# B&R Automation Studio project BR_Lab4
Automation Studio 4.5.2.102

## Configuration Real

### Task classes (Cpu.sw)
```
Cyclic#1:
  SDCAxisCtr <- SDCAxisCtrl_X.prg
DataObjects: Arnc0sys
NcDataObjects: gAxis01a <- gAxis01obj.gAxis01a.dob, gAxis01i <- gAxis01obj.gAxis01i.dob
Binaries: TCData, Acp10map1, acp10cfg, Acp10map, arconfig, User, Role, sysconf, iomap, asfw, ashwd, arnc0cfg, Arnc0map
Libraries: Acp10sdc, Library, Acp10man, Acp10_MC, sys_lib, brsystem, asstring, powerlnk, asieccon, AsMath, Arnc0man, DataObj, AsArLog, FileIO, AsArProf, AsMem, Runtime, astime, Acp10par, NcGlobal, asiotime
```

### IoMap.iom - 4PP065_0571_P74/IoMap.iom
```iecst
VAR_CONFIG
	::SDCAxisCtr:pwm_period AT %QW."X20MM4456".PeriodDurationPWM;
	::SDCAxisCtr:coil_pwm_value AT %QW."X20MM4456".PulseWidthCurrentPWM04;
	::SDCAxisCtr:axis_X.pwm_value AT %QW."X20MM4456".PulseWidthCurrentPWM01;
	::SDCAxisCtr:axis_X.reset_error AT %QX."X20MM4456".ClearError01;
	::SDCAxisCtr:axis_X.reset_counter AT %QX."X20MM4456".ResetCounter01;
	::SDCAxisCtr:axis_X.counter AT %IW."X20MM4456".Counter01;
	::SDCAxisCtr:coil_powered AT %IX."X20DI9371".DigitalInput01;
	::SDCAxisCtr:axis_X.endswitch_a_reached AT %IX."X20MM4456".StatusInput03;
	::SDCAxisCtr:axis_X.endswitch_b_reached AT %IX."X20MM4456".StatusInput04;
	::SDCAxisCtr:posEnable.enable AT %IX."X20DI9371".DigitalInput02; (*Insert your comment here...*)
	::SDCAxisCtr:posEnableRight.enable AT %IX."X20DI9371".DigitalInput03; (*Insert your comment here...*)
END_VAR
```

## Logical view

### Global.var - Global variables
```iecst
VAR
	AxisX_DrvIf : SdcDrvIf16_typ := (0);
	AxisX_EncIf : SdcEncIf16_typ := (0);
	AxisX_DiDoIf : SdcDiDoIf_typ := (0);
	AxisX_HW : SdcHwCfg_typ := (0);
	fb_regulator : FB_Regulator;
	iPosHwEnd : BOOL := FALSE;
	iNegHwEnd : BOOL := FALSE;
END_VAR
```

### Program Logical/SDCAxisCtrl_X (ANSIC)

#### Variables.var
```iecst
VAR
	axis_X : FB_Axis;
	coil_powered : BOOL := FALSE;
	coil_pwm_value : {REDUND_UNREPLICABLE} INT := 200;
	pwm_period : {REDUND_UNREPLICABLE} UINT := 200;
	Already_Homed : BOOL := FALSE;
	k : INT := 0;
	posEnable : Pos := (0);
	posEnableRight : Pos := (0);
END_VAR
```

#### Main.c
```c
#include <bur/plctypes.h>

#ifdef _DEFAULT_INCLUDES
 #include <AsDefault.h>
#endif

void increase_counters(void);

void _INIT ProgramInit(void)
{
 AxisX_HW.EncIf1_Typ = ncSDC_ENC16;
 AxisX_HW.DiDoIf_Typ = ncSDC_DIDO;
 AxisX_HW.DrvIf_Typ = ncSDC_DRVSERVO16;

 strcpy(AxisX_HW.EncIf1_Name, "AxisX_EncIf");
 strcpy(AxisX_HW.DrvIf_Name, "AxisX_DrvIf");
 strcpy(AxisX_HW.DiDoIf_Name, "AxisX_DiDoIf");

 AxisX_EncIf.iEncOK = 1;
 AxisX_DrvIf.iDrvOK = 1;
 AxisX_DrvIf.iStatusEnable = 1;
 AxisX_DiDoIf.iDriveReady = 1;

 fb_controller.dt = 0.002;
 fb_controller.k_i = 0.16;
 fb_controller.k_p = 0.0064;
 fb_controller.max_abs_value = 24.0;

 pwm_period = 200;
}

void _CYCLIC ProgramCyclic(void)
{
 if (posEnable.enable) {
  // axis_X.endswitch_a_reached = 1;
  AxisX_DrvIf.oSetPos = -10000;
 } else if (posEnableRight.enable) {
  AxisX_DrvIf.oSetPos = 10000;
 }
 FB_Axis(&axis_X);
 coil_pwm_value = coil_powered ? 32767 : 0;

 increase_counters();

 AxisX_EncIf.iActTime = (INT) AsIOTimeCyclicStart();
 AxisX_EncIf.iActPos = axis_X.counter;
 AxisX_DiDoIf.iPosHwEnd = axis_X.endswitch_b_reached;
 AxisX_DiDoIf.iNegHwEnd = axis_X.endswitch_a_reached;
 fb_controller.in = AxisX_DrvIf.oSetPos;

 if((fb_controller.in<min_task)&&(fb_controller.in>(-min_task))) fb_controller.in = 0;
 fb_controller.in = fb_controller.in * 6500/32767 - axis_X.speed;

 FB_Controller(&fb_controller);

 axis_X.pwm_value = fb_controller.out / 24.0 * 32767;
}

void increase_counters(void)
{
 AxisX_EncIf.iLifeCnt++;
 AxisX_DiDoIf.iLifeCntDriveEnable++;
 AxisX_DiDoIf.iLifeCntDriveReady++;
 AxisX_DiDoIf.iLifeCntNegHwEnd++;
 AxisX_DiDoIf.iLifeCntPosHwEnd++;
 AxisX_DiDoIf.iLifeCntReference++;
 AxisX_DrvIf.iLifeCnt++;
}

void _EXIT ProgramExit(void)
{
 // Insert code here

}
```

### Program Logical/SDCAxisCtrl_Y

#### Main.c
```c
#include <bur/plctypes.h>

#ifdef _DEFAULT_INCLUDES
 #include <AsDefault.h>
#endif

void _INIT ProgramInit(void)
{
 AxisY_HW.EncIf1_Typ = ncSDC_ENC16;
 AxisY_HW.DiDoIf_Typ = ncSDC_DIDO;
 AxisY_HW.DrvIf_Typ = ncSDC_DRVSERVO16;

 strcpy(AxisY_HW.EncIf1_Name, "AxisY_EncIf");
 strcpy(AxisY_HW.DrvIf_Name, "AxisY_DrvIf");
 strcpy(AxisY_HW.DiDoIf_Name, "AxisY_DiDoIf");

 AxisY_EncIf.iEncOK = 1;
 AxisY_DrvIf.iDrvOK = 1;
 AxisY_DrvIf.iStatusEnable = 1;
 AxisY_DiDoIf.iDriveReady = 1;

 fb_controller.dt = 0.002;
 fb_controller.k_i = 0.16;
 fb_controller.k_p = 0.0064;
 fb_controller.max_abs_value = 24.0;

 pwm_period = 200;

}

void _CYCLIC ProgramCyclic(void)
{
 if (posEnable.enable) {
  // axis_X.endswitch_a_reached = 1;
  AxisY_DrvIf.oSetPos = -10000;
 } else if (posEnableRight.enable) {
  AxisY_DrvIf.oSetPos = 10000;
 }
 FB_Axis(&axis_Y);
 coil_pwm_value = coil_powered ? 32767 : 0;

 increase_counters();

 AxisY_EncIf.iActTime = (INT) AsIOTimeCyclicStart();
 AxisY_EncIf.iActPos = axis_Y.counter;
 AxisY_DiDoIf.iPosHwEnd = axis_Y.endswitch_b_reached;
 AxisY_DiDoIf.iNegHwEnd = axis_Y.endswitch_a_reached;
 fb_controller.in = AxisY_DrvIf.oSetPos;

 if((fb_controller.in<min_task)&&(fb_controller.in>(-min_task))) fb_controller.in = 0;
 fb_controller.in = fb_controller.in * 6500/32767 - axis_Y.speed;

 FB_Controller(&fb_controller);

 axis_Y.pwm_value = fb_controller.out / 24.0 * 32767;
}

void increase_counters(void)
{
 AxisY_EncIf.iLifeCnt++;
 AxisY_DiDoIf.iLifeCntDriveEnable++;
 AxisY_DiDoIf.iLifeCntDriveReady++;
 AxisY_DiDoIf.iLifeCntNegHwEnd++;
 AxisY_DiDoIf.iLifeCntPosHwEnd++;
 AxisY_DiDoIf.iLifeCntReference++;
 AxisY_DrvIf.iLifeCnt++;
}

void _EXIT ProgramExit(void)
{
 // Insert code here

}
```

### Program Logical/SDCAxisCtrl_Z

#### Main.c
```c
#include <bur/plctypes.h>

#ifdef _DEFAULT_INCLUDES
 #include <AsDefault.h>
#endif

void _INIT ProgramInit(void) {

 AxisZ_HW.EncIf1_Typ = ncSDC_ENC16;
 AxisZ_HW.DiDoIf_Typ = ncSDC_DIDO;
 AxisZ_HW.DrvIf_Typ = ncSDC_DRVSERVO16;

 strcpy(AxisZ_HW.EncIf1_Name, "AxisZ_EncIf");
 strcpy(AxisZ_HW.DrvIf_Name, "AxisZ_DrvIf");
 strcpy(AxisZ_HW.DiDoIf_Name, "AxisZ_DiDoIf");

 AxisZ_EncIf.iEncOK = 1;
 AxisZ_DrvIf.iDrvOK = 1;
 AxisZ_DrvIf.iStatusEnable = 1;
 AxisZ_DiDoIf.iDriveReady = 1;

 fb_controller.dt = 0.002;
 fb_controller.k_i = 0.16;
 fb_controller.k_p = 0.0064;
 fb_controller.max_abs_value = 24.0;

 pwm_period = 200;
}

void _CYCLIC ProgramCyclic(void)
{
 if (posEnable.enable) {
  // axis_X.endswitch_a_reached = 1;
  AxisZ_DrvIf.oSetPos = -10000;
 } else if (posEnableRight.enable) {
  AxisZ_DrvIf.oSetPos = 10000;
 }
 FB_Axis(&axis_Z);
 coil_pwm_value = coil_powered ? 32767 : 0;

 increase_counters();

 AxisZ_EncIf.iActTime = (INT) AsIOTimeCyclicStart();
 AxisZ_EncIf.iActPos = axis_Z.counter;
 AxisZ_DiDoIf.iPosHwEnd = axis_Z.endswitch_b_reached;
 AxisZ_DiDoIf.iNegHwEnd = axis_Z.endswitch_a_reached;
 fb_controller.in = AxisZ_DrvIf.oSetPos;

 if((fb_controller.in<min_task)&&(fb_controller.in>(-min_task))) fb_controller.in = 0;
 fb_controller.in = fb_controller.in * 6500/32767 - axis_Z.speed;

 FB_Controller(&fb_controller);

 axis_Z.pwm_value = fb_controller.out / 24.0 * 32767;

}

void increase_counters(void)
{
 AxisZ_EncIf.iLifeCnt++;
 AxisZ_DiDoIf.iLifeCntDriveEnable++;
 AxisZ_DiDoIf.iLifeCntDriveReady++;
 AxisZ_DiDoIf.iLifeCntNegHwEnd++;
 AxisZ_DiDoIf.iLifeCntPosHwEnd++;
 AxisZ_DiDoIf.iLifeCntReference++;
 AxisZ_DrvIf.iLifeCnt++;

}

void _EXIT ProgramExit(void)
{
 // Insert code here

}
```

Listed in the project but not available here: Logical/Global.typ, Logical/Libraries, Logical/Types.typ, Logical/gAxis01obj
